KUKA KRL program: SystemPurge.src, SystemPurge.dat

--- SystemPurge.src ---
&ACCESS RVP
&REL 23
&PARAM EDITMASK = *
&PARAM TEMPLATE = C:\KRC\Roboter\Template\vorgabe
&PARAM DISKPATH = KRC:\R1\Program\CNCRobotics\CEAD
DEF SystemPurge( )
DECL INT _nAns
;FOLD INI;%{PE}
  ;FOLD BASISTECH INI
    GLOBAL INTERRUPT DECL 3 WHEN $STOPMESS==TRUE DO IR_STOPM ( )
    INTERRUPT ON 3
GLOBAL INTERRUPT DECL 4 WHEN bCeadInterrupt==TRUE DO CeadInterrupt ( )
INTERRUPT ON 4
    BAS (#INITMOV,0 )
  ;ENDFOLD (BASISTECH INI)
  ;FOLD USER INI
    ;Make your modifications here

  ;ENDFOLD (USER INI)
  ;ENDFOLD (INI)

;************************************************
;              CNC Robotics Ltd
;************************************************
;     Contact: helpdesk@cncrobotics.co.uk
;     Date: 26/09/23
;     Version: 0.18.51
;************************************************
; Description: Routine to purge the extruder of
; all material and run purge compund through to
; clear out the extruder.
;************************************************

;Start by moving robot to the home position
HomePosition()

;Check with operator that they have closed the slide to stop material going from the dryer to the hoppper
MsgDialog(_nAns,"Please close the dryer slide to stop more material coming through.","CEAD",,,,,,,,"OK", FALSE, nCeadMsg + 10, E_spsMsgOpt)

;Prevent system from stopping when hopper is empty
oEmptyHopperBypass = FALSE

;Motion to move the robot to the purge position

;Set extruder perameters
rPumpTime = 15	;Time(seconds) pump will pull material to the hopper
rShotSize = 1.0 ;Time(seconds) the pinch valve will open, allowing material through
SetPelletSource (#DRYER) ;Set the source of material as the dryer

SetHeatZones (rTempSet1,rTempSet2,rTempSet3,rTempSet4) ;Set heatzones to previous values

TransportOn()  ;Start transport system
WaitForReady() ;Wait for heatzsones up to temperature and 10 min timer

RotationOn()   ;Start extruding
SetScrewSpeed(50);Set extruder speed to 50RPM

;Extrude until the hopper is empty of material, then for another 2 mins to fully clear the extruder
WAIT FOR iTransportWarning
WAIT SEC 120

;Stop Extruding
SetScrewSpeed(0)
RotationOff()

;Warn the operator that they must have purge compound in the base unit storage
MsgDialog(_nAns,"Please ensure cabinet storage contains purge compound now.","CEAD",,,,,,,,"OK", FALSE, nCeadMsg + 11, E_spsMsgOpt)

;Change the material selection to draw from the cabinet storage
SetPelletSource (#INTERNAL_CABINET)
;Update heatzones to settings for purge compound and wait for system ready
SetHeatZones (180,190,200,200)
WaitForReady()

;Start extrusion
RotationOn()
SetScrewSpeed(50)

WAIT SEC 300 ;Wait 5 minutes until purge compound is in extruder

_nAns=0
WHILE _nAns<>1
	;Check if system is successfully purged
	MsgDialog(_nAns,"Has the system been purged successfully.","CEAD",,,,,,,"No","Yes", FALSE, nCeadMsg + 12, E_spsMsgOpt)
	IF _nAns <> 1 THEN
		WAIT SEC 120 ;If not fully purged, extrude for another 2 mins
	ENDIF
ENDWHILE

;Stop Extruding
SetScrewSpeed(0)
FinishPrint()

;Return to home
HomePosition()

END

--- SystemPurge.dat ---
&ACCESS RVP
&REL 23
&PARAM EDITMASK = *
&PARAM TEMPLATE = C:\KRC\Roboter\Template\vorgabe
&PARAM DISKPATH = KRC:\R1\Program\CNCRobotics\CEAD
DEFDAT  SYSTEMPURGE
;FOLD EXTERNAL DECLARATIONS;%{PE}%MKUKATPBASIS,%CEXT,%VCOMMON,%P
;FOLD BASISTECH EXT;%{PE}%MKUKATPBASIS,%CEXT,%VEXT,%P
EXT  BAS (BAS_COMMAND  :IN,REAL  :IN )
DECL INT SUCCESS
;ENDFOLD (BASISTECH EXT)
;FOLD USER EXT;%{E}%MKUKATPUSER,%CEXT,%VEXT,%P
;Make your modifications here

;ENDFOLD (USER EXT)
;ENDFOLD (EXTERNAL DECLARATIONS)
DECL BASIS_SUGG_T LAST_BASIS={POINT1[] "P3                      ",POINT2[] "P3                      ",CP_PARAMS[] "CPDAT0                  ",PTP_PARAMS[] "PDAT4                   ",CONT[] "C_DIS                   ",CP_VEL[] "2.0                     ",PTP_VEL[] "20                      ",SYNC_PARAMS[] "SYNCDAT                 ",SPL_NAME[] "S0                      ",A_PARAMS[] "ADAT0                   "}
DECL E6POS XP1={X 1044.07520,Y -1448.90295,Z 2604.21387,A -0.207003787,B 32.7573776,C 0.167719990,S 22,T 27,E1 1450.01270,E2 0.0,E3 0.0,E4 0.0,E5 0.0,E6 0.0}
DECL FDAT FP1={TOOL_NO 0,BASE_NO 0,IPO_FRAME #BASE,POINT2[] " "}
DECL PDAT PPDAT1={VEL 20.0000,ACC 100.000,APO_DIST 500.000,APO_MODE #CDIS,GEAR_JERK 100.000,EXAX_IGN 0}
DECL MODULEPARAM_T LAST_TP_PARAMS={PARAMS[] "Kuka.PointName=P3; Kuka.FrameData.base_no=1; Kuka.FrameData.tool_no=1; Kuka.FrameData.ipo_frame=#BASE; Kuka.isglobalpoint=False; Kuka.MoveDataPtpName=PDAT5; Kuka.MovementDataPdat.apo_mode=#CDIS; Kuka.MovementDataPdat.apo_dist=500; Kuka.MovementData.vel=30; Kuka.MovementData.acc=100; Kuka.MovementData.exax_ign=0; Kuka.VelocityPtp=30; Kuka.BlendingEnabled=True; Kuka.CurrentCDSetIndex=0; Kuka.FrameData.point2=; Kuka.APXEnabled=False; Kuka.VelocityFieldEnabled=True; Kuka.ColDetectFieldEnabled=True; Kuka.MovementParameterFieldEnabled=True; Kuka.IsAngleEnabled=False    "}
DECL PDAT PPDAT2={VEL 20.0000,ACC 100.000,APO_DIST 500.000,APO_MODE #CDIS,GEAR_JERK 100.000,EXAX_IGN 0}
DECL E6POS XP2={X 985.740784,Y -188.071182,Z 195.024033,A -53.5795326,B 89.7479401,C -53.8516121,S 22,T 18,E1 1043.05981,E2 0.0,E3 0.0,E4 0.0,E5 0.0,E6 0.0}
DECL FDAT FP2={TOOL_NO 1,BASE_NO 1,IPO_FRAME #BASE,POINT2[] " "}
DECL PDAT PPDAT3={VEL 100.000,ACC 100.000,APO_DIST 500.000,APO_MODE #CDIS,GEAR_JERK 50.0000,EXAX_IGN 0}
DECL E6POS XP3={X 985.277466,Y -128.016129,Z 601.188782,A -55.3659096,B 89.7469635,C -55.6446457,S 22,T 27,E1 1043.05981,E2 0.0,E3 0.0,E4 0.0,E5 0.0,E6 0.0}
DECL FDAT FP3={TOOL_NO 1,BASE_NO 1,IPO_FRAME #BASE,POINT2[] " "}
DECL PDAT PPDAT4={VEL 30.0000,ACC 100.000,APO_DIST 500.000,APO_MODE #CDIS,GEAR_JERK 50.0000,EXAX_IGN 0}
DECL PDAT PPDAT5={VEL 30.0000,ACC 100.000,APO_DIST 500.000,APO_MODE #CDIS,GEAR_JERK 100.000,EXAX_IGN 0}
DECL PDAT PPDAT6={VEL 30.0000,ACC 100.000,APO_DIST 500.000,APO_MODE #CDIS,GEAR_JERK 100.000,EXAX_IGN 0}
DECL PDAT PPDAT9={VEL 30.0000,ACC 100.000,APO_DIST 500.000,APO_MODE #CDIS,GEAR_JERK 100.000,EXAX_IGN 0}
DECL PDAT PPDAT10={VEL 30.0000,ACC 100.000,APO_DIST 500.000,APO_MODE #CDIS,GEAR_JERK 100.000,EXAX_IGN 0}
DECL LDAT LCPDAT5={VEL 0.500000,ACC 100.000,APO_DIST 500.000,APO_FAC 50.0000,AXIS_VEL 100.000,AXIS_ACC 100.000,ORI_TYP #VAR,CIRC_TYP #BASE,JERK_FAC 50.0000,GEAR_JERK 100.000,EXAX_IGN 0,CB {AUX_PT {ORI #CONSIDER,E1 #CONSIDER,E2 #CONSIDER,E3 #CONSIDER,E4 #CONSIDER,E5 #CONSIDER,E6 #CONSIDER},TARGET_PT {ORI #INTERPOLATE,E1 #INTERPOLATE,E2 #INTERPOLATE,E3 #INTERPOLATE,E4 #INTERPOLATE,E5 #INTERPOLATE,E6 #INTERPOLATE}}}
DECL LDAT LCPDAT6={VEL 0.500000,ACC 100.000,APO_DIST 500.000,APO_FAC 50.0000,AXIS_VEL 100.000,AXIS_ACC 100.000,ORI_TYP #VAR,CIRC_TYP #BASE,JERK_FAC 50.0000,GEAR_JERK 100.000,EXAX_IGN 0,CB {AUX_PT {ORI #CONSIDER,E1 #CONSIDER,E2 #CONSIDER,E3 #CONSIDER,E4 #CONSIDER,E5 #CONSIDER,E6 #CONSIDER},TARGET_PT {ORI #INTERPOLATE,E1 #INTERPOLATE,E2 #INTERPOLATE,E3 #INTERPOLATE,E4 #INTERPOLATE,E5 #INTERPOLATE,E6 #INTERPOLATE}}}
ENDDAT
